// Mitsubishi GX Works2 project: 241129_ex1   PLC: Q02U

PROGRAM MAIN
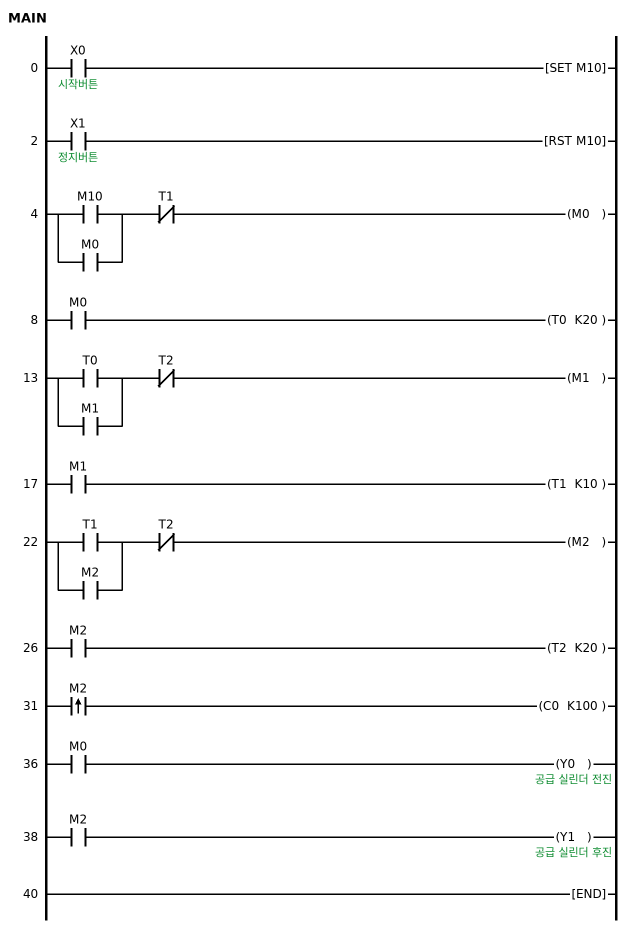
0     LD      X0  ; 시작버튼
      SET     M10
2     LD      X1  ; 정지버튼
      RST     M10
4     LD      M10
      OR      M0
      ANI     T1
      OUT     M0
8     LD      M0
      OUT     T0 K20
13    LD      T0
      OR      M1
      ANI     T2
      OUT     M1
17    LD      M1
      OUT     T1 K10
22    LD      T1
      OR      M2
      ANI     T2
      OUT     M2
26    LD      M2
      OUT     T2 K20
31    LDP     M2
      OUT     C0 K100
36    LD      M0
      OUT     Y0  ; 공급 실린더 전진
38    LD      M2
      OUT     Y1  ; 공급 실린더 후진
40    END
END_PROGRAM

// device comments not shown above
X2  ; 긴급정지버튼
X3  ; 공급센서
X4  ; 물체확인센서
X5  ; 금속확인센서
X6  ; 공급실린더ForwardLS
X7  ; 공급실린더BackwardLS
X8  ; 가공실린더ForwardLS
X9  ; 가공실린더BackwardLS
X0A  ; 송출실린더ForwardLS
X0B  ; 송출실린더BackwardLS
X0C  ; 배출실린더ForwardLS
X0D  ; 배출실린더BackwardLS
Y2  ; 가공 실린더 전진
Y3  ; 가공 실린더 후진
Y4  ; 송출 실린더 전진
Y5  ; 송출 실린더 후진
Y6  ; 배출 실린더 전진
Y7  ; 배출 실린더 후진
Y8  ; 컨베이어 CW
Y9  ; 컨베이어 CCW
Y0A  ; 컨베이어 STOP
Y0B  ; 램프 RED
Y0C  ; 램프 YELLOW
Y0D  ; 램프 GREEN
